# B&R Automation Studio project lab3
Automation Studio 

## Configuration Real

CPU 4PP065.0571-P74, AutomationRuntime D4.52, Build 4.1.2, Vc V4.52.0, Safety 1.6

### Task classes (Cpu.sw)
```
Cyclic#1 (cycle 2000 us, tolerance 0 us):
  ncsdcctrl <- ncsdcctrl.prg
  SDCAxisCtr <- SDCAxisCtrl_X.prg
  SDCAxisCt2 <- SDCAxisCtrl_Z.prg
  SDCAxisCt1 <- SDCAxisCtrl_Y.prg
Cyclic#2:
  User_Inter <- User_Interface.prg
DataObjects: Arnc0sys, Acp10sys
NcDataObjects: AxisInit <- AxisInit.dob, gAxis03a <- gAxis03obj.gAxis03a.dob, gAxis03i <- gAxis03obj.gAxis03i.dob, AxisApt <- AxisApt.dob, gmcipsys <- GmcIpConfig.gmcipsys.dob, gmcipusm <- GmcIpUserConfig.gmcipusm.dob, gmciplbr <- GmcIpConfig.gmciplbr.dob, gmcipvar <- GmcIpUserConfig.gmcipvar.dob, gmcipcbr <- GmcIpConfig.gmcipcbr.dob, gmcipubr <- GmcIpUserConfig.gmcipubr.dob, gmciplsm <- GmcIpConfig.gmciplsm.dob, gmcipui <- GmcIpUserConfig.gmcipui.dob, gmcipcsm <- GmcIpConfig.gmcipcsm.dob, gmcipuc <- GmcIpUserConfig.gmcipuc.dob, gmcipcfg <- GmcIpConfig.gmcipcfg.dob, gmcipfub <- GmcIpUserConfig.gmcipfub.dob, gmcipiec <- GmcIpConfig.gmcipiec.dob, gmcipus <- GmcIpUserConfig.gmcipus.dob, gmciplog <- GmcIpConfig.gmciplog.dob, gmcipfun <- GmcIpUserConfig.gmcipfun.dob, gmcipesm <- GmcIpConfig.gmcipesm.dob, gmcipmxd <- GmcIpConfig.gmcipmxd.dob, gmcipmx <- GmcIpConfig.gmcipmx.dob, CncInit <- CncInit.dob, CncProg1 <- CncProg1.dob, CncProg <- CncProg.dob
VcDataObjects: Visu <- Visu.dob
Binaries: TCData, vccbtn, arialbd, vcmgr, vcfile, vccnum, vcpfpp30, vcfntttf, vctcal, vcdsloc, vcgclass, vcpfmtcx, vcbclass, udbdef, arial, Visu03, vcalarm, Visu01, vcptelo, vcpdpp30, vcrt, vcshared, Visu02, vcctext, vcdsint, vcpdsw, vccovl, arconfig, User, Role, sysconf, iomap, asfw, ashwd, ashwac, Acp10map1, acp10cfg, Acp10map, arnc0cfg, Arnc0map
Libraries: Acp10sdc, Library, Acp10man, Acp10_MC, sys_lib, brsystem, asstring, AsMath, Arnc0man, DataObj, AsArLog, FileIO, AsArProf, AsMem, Runtime, astime, Acp10par, NcGlobal, Acp10sim, powerlnk, asieccon, asiotime, vcresman, operator
```

### Hardware
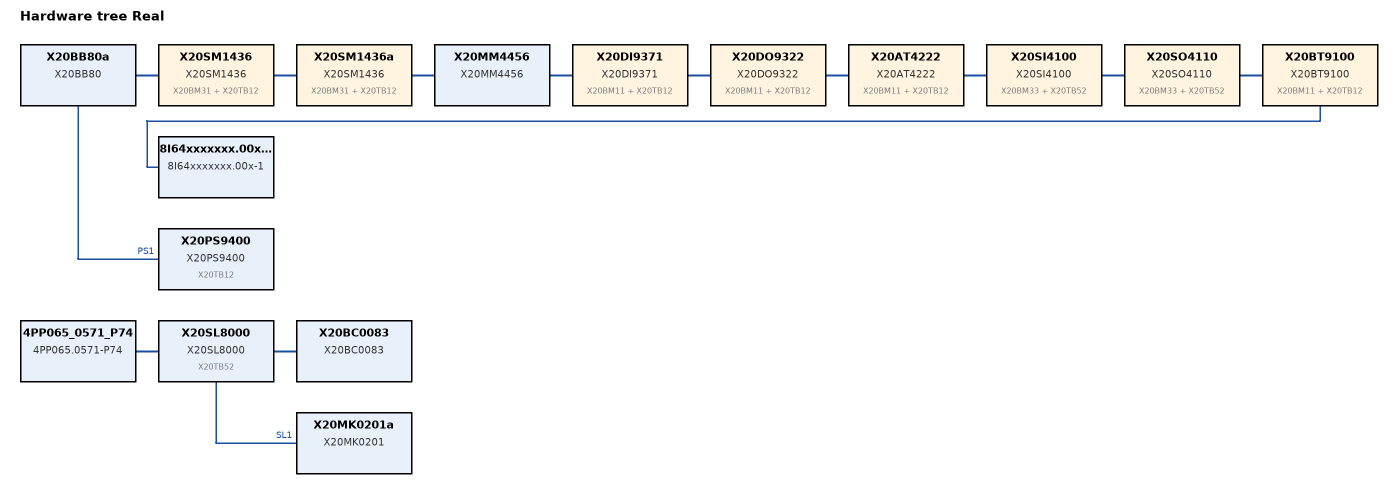
```
4PP065_0571_P74 : 4PP065.0571-P74 v1.1.2.0
  Connector IF4:
    Channel1
    ChannelID1 = McAcpBroadcast
    ChannelType1 = OCTET[96]
  Connector IF5:
    ActivateDevice = 1
    Mode = Manual
    InternetAddress = 10.0.1.14
    SubnetMask = 255.255.255.0
  ConfigurationID = labBR
  TimerDeviceType = EPLX2X
  TimerDevice = 4PP065_0571_P74.IF4
  TaskClassIdleTime = 2000
  Cyclic1Duration = 2000
  Cyclic1Tolerance = 0
  Cyclic1Output = 1
  Cyclic3Tolerance = 0
  VcObjectName = Visu
8I64xxxxxxx.00x-1 : 8I64xxxxxxx.00x-1 v1.3.9.1  [X2X1 -> X20BT9100.X2X1 [Cable Type=X2XCable, Length=10, Version=1.0.0.2]]
  BothEndSwitchesAreNormallyOpen_r1 = on
  QuickStopIsNormallyOpen_r1 = on
X20AT4222 : X20AT4222 v1.2.3.0  [SS1 -> X20TB12f.SS; SL -> X20BM11c.SL1]
X20BB80a : X20BB80 v1.0.2.0
X20BC0083 : X20BC0083 v2.7.0.0  [PLK1 -> X20SL8000.PLK2 (NodeNumber=2) [Cable Type=PowerlinkCable, Length=10, Version=1.0.0.2]; SL -> X20BB80a.SL1]
X20BM11a : X20BM11 v1.0.0.1  [X2X1 -> X20MM4456.X2X2]
X20BM11b : X20BM11 v1.0.0.1  [X2X1 -> X20BM11a.X2X2]
X20BM11c : X20BM11 v1.0.0.1  [X2X1 -> X20BM11b.X2X2]
X20BM11d : X20BM11 v1.0.0.1  [X2X1 -> X20BM33b.X2X2]
X20BM31a : X20BM31 v1.0.0.1  [X2X1 -> X20BB80a.IF1]
X20BM31b : X20BM31 v1.0.0.1  [X2X1 -> X20BM31a.X2X2]
X20BM33a : X20BM33 v1.0.0.4  [X2X1 -> X20BM11c.X2X2]
X20BM33b : X20BM33 v1.0.0.4  [X2X1 -> X20BM33a.X2X2]
X20BT9100 : X20BT9100 v1.0.3.0  [SS1 -> X20TB12g.SS; SL -> X20BM11d.SL1]
X20DI9371 : X20DI9371 v1.0.2.0  [SS1 -> X20TB12d.SS; SL -> X20BM11a.SL1]
X20DO9322 : X20DO9322 v1.0.3.0  [SS1 -> X20TB12e.SS; SL -> X20BM11b.SL1]
X20MK0201a : X20MK0201 v1.0.0.0 (Disabled=true)  [SL -> X20SL8000.SL1]
X20MM4456 : X20MM4456 v1.1.5.0  [X2X1 -> X20BM31b.X2X2]
X20PS9400 : X20PS9400 v1.0.2.4  [SS1 -> X20TB12b.SS; PS -> X20BB80a.PS1]
X20SI4100 : X20SI4100 v1.10.1.1  [SS1 -> X20TB52b.SS; SL -> X20BM33a.SL1]
X20SL8000 : X20SL8000 v1.6.5.1 (Disabled=true)  [PLK1 -> 4PP065_0571_P74.IF4 (NodeNumber=1) [Cable Type=PowerlinkCable, Length=10, Version=1.0.0.2]; PLK2 -> X20BC0083.PLK1 (NodeNumber=1) [Cable Type=PowerlinkCable, Length=10, Version=1.0.0.2]; SS1 -> X20TB52a.SS]
  SafeProject = SafeLOGIC-1
X20SM1436 : X20SM1436 v1.4.2.1  [SS1 -> X20TB12a.SS; SL -> X20BM31a.SL1]
X20SM1436a : X20SM1436 v1.4.2.1  [SS1 -> X20TB12c.SS; SL -> X20BM31b.SL1]
X20SO4110 : X20SO4110 v1.10.1.1  [SS1 -> X20TB52c.SS; SL -> X20BM33b.SL1]
  SafeLogicID = 2
  SafeModuleID = 3
X20TB12a : X20TB12 v1.0.0.0
X20TB12b : X20TB12 v1.0.0.0
X20TB12c : X20TB12 v1.0.0.0
X20TB12d : X20TB12 v1.0.0.0
X20TB12e : X20TB12 v1.0.0.0
X20TB12f : X20TB12 v1.0.0.0
X20TB12g : X20TB12 v1.0.0.0
X20TB52a : X20TB52 v1.0.0.1 (Disabled=true)
X20TB52b : X20TB52 v1.0.0.1
X20TB52c : X20TB52 v1.0.0.1
```

## Configuration Simulation

### Task classes (Cpu.sw)
```
Cyclic#1:
  SDCAxisCtr <- SDCAxisCtrl_X.prg
DataObjects: Acp10sys
NcDataObjects: AxisApt <- AxisApt.dob, AxisInit <- AxisInit.dob, acp10etxen <- acp10etxen.dob
Binaries: TCData, ashwd, sysconf, asfw, arconfig, iomap, Acp10map, Acp10map1, arnc0cfg, acp10cfg
Libraries: AsIecCon, astime, Acp10sdc, Acp10man, Acp10par, NcGlobal, asstring, AsIOTime, Acp10_MC, brsystem, sys_lib, Runtime, Acp10sim, fileio, powerlnk, Library
```

## Logical view

Binary libraries used (declarations not repeated): Runtime, Operator, AsIecCon, astime, asstring, AsIOTime, brsystem, sys_lib, AsMath, DataObj, AsArLog, FileIO, AsArProf, AsMem, Acp10man, Acp10par, NcGlobal, Acp10sim, Acp10_MC, Acp10sdc, Arnc0man 5.02.1

### Global.var
```iecst
VAR
	Trajectory : FB_Trajectory := (0); (*Переменная типа Функциональный блок управления УРТК*)
	Move_axis : FB_move := (0); (*Переменная типа Функциональный блок движения оси*)
	Power_home : FB_power := (0); (*Переменная типа Функциональный блок запуска и референсирование осей*)
	AxisX : ACP10AXIS_typ := (0); (*Ось X*)
	AxisX_EncIf : SdcEncIf16_typ := (0);
	AxisX_DrvIf : SdcDrvIf16_typ := (0);
	AxisX_DiDoIf : SdcDiDoIf_typ := (0);
	AxisX_HW : SdcHwCfg_typ := (0);
	AxisY : ACP10AXIS_typ := (0); (*Ось Y*)
	AxisY_EncIf : SdcEncIf16_typ := (0);
	AxisY_DrvIf : SdcDrvIf16_typ := (0);
	AxisY_DiDoIf : SdcDiDoIf_typ := (0);
	AxisY_HW : SdcHwCfg_typ := (0);
	AxisZ : ACP10AXIS_typ := (0); (*Ось Z*)
	AxisZ_EncIf : SdcEncIf16_typ := (0);
	AxisZ_DrvIf : SdcDrvIf16_typ := (0);
	AxisZ_DiDoIf : SdcDiDoIf_typ := (0);
	AxisZ_HW : SdcHwCfg_typ := (0);
	gAxis01 : ACP10AXIS_typ := (0);
	gAxis02 : ACP10AXIS_typ := (0);
	gAxisTest : ACP10AXIS_typ := (0);
	gAxisTest_HW : SdcHwCfg_typ := (0);
	gAxisTest_DrvIf : SdcDrvIf16_typ := (0);
	gAxisTest_DiDoIf : SdcDiDoIf_typ := (0);
	gAxisTest_ModuleOk : BOOL := 0;
	gAxis03 : ACP10AXIS_typ := (0);
	gAxis03_HW : SdcHwCfg_typ := (0);
	gAxis03_DrvIf : SdcDrvIf16_typ := (0);
	gAxis03_DiDoIf : SdcDiDoIf_typ := (0);
	gAxis03_ModuleOk : BOOL := 0;
	CNCsys : ARNC0CNC_typ;
END_VAR
```

### AxInitAcp10.ax
```
InitParameter (Version=5.2.1, NcSwId=ACP10)
  ACP10AXIS_typ:
    dig_in:
      level:
        reference = ncACTIV_HI
        pos_hw_end = ncACTIV_HI
        neg_hw_end = ncACTIV_HI
        trigger1 = ncACTIV_HI
        trigger2 = ncACTIV_HI
    encoder_if:
      parameter:
        count_dir = ncSTANDARD
        scaling:
          load:
            units = 3000
            rev_motor = 1
    limit:
      parameter:
        v_pos = 7500.0
        v_neg = 7500.0
        a1_pos = 10000.0
        a2_pos = 10000.0
        a1_neg = 10000.0
        a2_neg = 10000.0
        t_jolt = 0.0
        t_in_pos = 0.0
        pos_sw_end = 8388607
        neg_sw_end = -8388608
        ds_warning = 500.0
        ds_stop = 1000.0
        a_stop = 1.0E+30
        dv_stop = 0.0
        dv_stop_mode = ncOFF
    controller:
      mode = ncPOSITION
      position:
        kv = 10.0
        tn = 0.0
        t_predict = 0.04
        t_total = 0.04
        p_max = 10000.0
        i_max = 0.0
      speed:
        kv = 100.0
        tn = 0.04
        t_filter = 0.0
        isq_filter1:
          type = ncOFF
          a0 = 0.0
          a1 = 0.0
          b0 = 0.0
          b1 = 0.0
          b2 = 0.0
          c0_par_id = 0
          c1_par_id = 0
        isq_filter2:
          type = ncOFF
          a0 = 0.0
          a1 = 0.0
          b0 = 0.0
          b1 = 0.0
          b2 = 0.0
          c0_par_id = 0
          c1_par_id = 0
        isq_filter3:
          type = ncOFF
          a0 = 0.0
          a1 = 0.0
          b0 = 0.0
          b1 = 0.0
          b2 = 0.0
          c0_par_id = 0
          c1_par_id = 0
      uf:
        type = ncLINEAR
        auto_config = ncMOTOR_PAR
        u0 = 0.0
        un = 0.0
        fn = 50.0
        k_f_slip = 0.0
      ff:
        torque_load = 0.0
        torque_pos = 0.0
        torque_neg = 0.0
        kv_torque = 0.0
        inertia = 0.0
        t_filter_a = 0.0
    move:
      stop:
        parameter[0]:
          decel_ramp = ncA_LIMIT
          controller = ncON
        parameter[1]:
          decel_ramp = ncA_LIMIT
          controller = ncON
        parameter[2]:
          decel_ramp = ncA_LIMIT
          controller = ncON
        parameter[3]:
          decel_ramp = ncA_LIMIT
          controller = ncON
        quickstop:
          decel_ramp = ncA_LIMIT
          t_jolt = 0.0
        drive_error:
          decel_ramp = ncA_LIMIT
      homing:
        parameter:
          s = 0
          v_switch = 2000.0
          v_trigger = 1000.0
          a = 5000.0
          mode = ncDIRECT
          edge_sw = ncNEGATIVE
          start_dir = ncPOSITIVE
          trigg_dir = ncNEGATIVE
          ref_pulse = ncOFF
          fix_dir = ncOFF
          tr_s_block = 0.0
          torque_lim = 0.0
          ds_block = 0.0
          ds_stop = 0.0
      basis:
        parameter:
          v_pos = 6000.0
          v_neg = 6000.0
          a1_pos = 12000.0
          a2_pos = 12000.0
          a1_neg = 12000.0
          a2_neg = 12000.0
    message:
      text:
        parameter:
          format = ncBREAK
          columns = 80
          data_modul
```

- Data object Logical/CncInit (Cns) (no source held here)

- Data object Logical/CncProg (Cnc) (no source held here)

- Data object Logical/GmcIpConfig/gmcipsys (Cnc, version 5.02.1) (no source held here)

- Data object Logical/GmcIpConfig/gmciplbr (Cnc, version 5.02.1) (no source held here)

- Data object Logical/GmcIpConfig/gmcipcbr (Cnc, version 5.02.1) (no source held here)

- Data object Logical/GmcIpConfig/gmciplsm (Cnc, version 5.02.1) (no source held here)

- Data object Logical/GmcIpConfig/gmcipcsm (Cnc, version 5.02.1) (no source held here)

- Data object Logical/GmcIpConfig/gmcipcfg (Cnc, version 5.02.1) (no source held here)

- Data object Logical/GmcIpConfig/gmcipiec (Cnc, version 5.02.1) (no source held here)

- Data object Logical/GmcIpConfig/gmciplog (Cnc, version 5.02.1) (no source held here)

- Data object Logical/GmcIpConfig/gmcipesm (Cnc, version 5.02.1) (no source held here)

- Data object Logical/GmcIpConfig/gmcipmxd (Cnc, version 5.02.1) (no source held here)

- Data object Logical/GmcIpConfig/gmcipmx (Cnc, version 5.02.1) (no source held here)

- Data object Logical/GmcIpUserConfig/gmcipfub (Cnc, version 5.02.1) (no source held here)

- Data object Logical/GmcIpUserConfig/gmcipfun (Cnc, version 5.02.1) (no source held here)

- Data object Logical/GmcIpUserConfig/gmcipubr (Cnc, version 5.02.1) (no source held here)

- Data object Logical/GmcIpUserConfig/gmcipuc (Cnc, version 5.02.1) (no source held here)

### Library Logical/Libraries/Library (ANSIC)
Depends on: Runtime, Operator, AsIecCon, astime, asstring, AsIOTime, brsystem, sys_lib, AsMath, DataObj, AsArLog, FileIO, AsArProf, AsMem, Acp10man, Acp10par, NcGlobal, Acp10sim, Acp10_MC, Acp10sdc, Arnc0man

#### Types.typ
```iecst
TYPE
	T_State_Trajectory :
		(
		Idle_Trajectory,
		Done_Trajectory,
		side1,
		side2,
		side3,
		side4,
		PowerY,
		PowerZ,
		Stop_Trajectory
		);
	T_State_move :
		(
		Idle_move,
		Move,
		Done_move
		);
	T_State_power :
		(
		Idle,
		Power,
		Home,
		Done
		);
END_TYPE
```

#### Library.fun
```iecst
FUNCTION_BLOCK FB_Motor (*TODO: Add your comment here*) (*$GROUP=User,$CAT=User,$GROUPICON=User.png,$CATICON=User.png*)
	VAR_INPUT
		in : REAL;
	END_VAR
	VAR_OUTPUT
		out_w : REAL;
		out_phi : REAL;
	END_VAR
	VAR
		k_e : REAL;
		T_m : REAL;
		dt : REAL;
		integrator : FB_Integrator;
		integrator_phi : FB_Integrator;
	END_VAR
END_FUNCTION_BLOCK

FUNCTION_BLOCK FB_Integrator (*TODO: Add your comment here*) (*$GROUP=User,$CAT=User,$GROUPICON=User.png,$CATICON=User.png*)
	VAR_INPUT
		in : REAL;
		dt : REAL;
	END_VAR
	VAR_OUTPUT
		out : REAL;
	END_VAR
	VAR
		state : REAL := 0.0;
	END_VAR
END_FUNCTION_BLOCK

FUNCTION_BLOCK FB_Controller (* *) (*$GROUP=User,$CAT=User,$GROUPICON=User.png,$CATICON=User.png*)
	VAR_INPUT
		in : REAL;
	END_VAR
	VAR_OUTPUT
		out : REAL;
	END_VAR
	VAR
		k_i : REAL;
		sum : REAL;
		k_p : REAL;
		dt : REAL;
		max_abs_value : REAL;
		integrator : FB_Integrator;
		last_sum : REAL;
	END_VAR
END_FUNCTION_BLOCK

FUNCTION_BLOCK FB_Endswitch (*TODO: Add your comment here*) (*$GROUP=User,$CAT=User,$GROUPICON=User.png,$CATICON=User.png*)
	VAR_INPUT
		in : REAL;
		neg_value : REAL;
		pos_value : REAL;
	END_VAR
	VAR_OUTPUT
		neg_reached : BOOL;
		pos_reached : BOOL;
	END_VAR
END_FUNCTION_BLOCK

FUNCTION_BLOCK FB_Axis (*TODO: Add your comment here*) (*$GROUP=User,$CAT=User,$GROUPICON=User.png,$CATICON=User.png*)
	VAR_INPUT
		reset_error : BOOL;
		endswitch_a_reached : BOOL;
		endswitch_b_reached : BOOL;
		pwm_percentage : SINT;
	END_VAR
	VAR_OUTPUT
		reset_counter : BOOL;
		pwm_value : INT;
	END_VAR
	VAR_OUTPUT RETAIN
		counter : INT;
	END_VAR
	VAR_OUTPUT
		speed : REAL;
	END_VAR
	VAR
		last_counter : INT;
	END_VAR
END_FUNCTION_BLOCK

{REDUND_ERROR} FUNCTION_BLOCK FB_power (*Функциональный блок запуска и референсирование осей*) (*$GROUP=User,$CAT=User,$GROUPICON=User.png,$CATICON=User.png*)
	VAR_INPUT
		State : T_State_power;
		Power : MC_Power;
		Home : MC_Home;
		Axis : UDINT;
		enable : BOOL;
	END_VAR
	VAR_OUTPUT
		done : BOOL;
	END_VAR
END_FUNCTION_BLOCK

{REDUND_ERROR} FUNCTION_BLOCK FB_move (*Функциональный блок движения оси*) (*$GROUP=User,$CAT=User,$GROUPICON=User.png,$CATICON=User.png*)
	VAR_INPUT
		Axis : UDINT;
		enable : BOOL;
		Move : MC_MoveAdditive;
		length : REAL;
	END_VAR
	VAR_OUTPUT
		done : BOOL;
	END_VAR
	VAR
		State : T_State_move;
	END_VAR
END_FUNCTION_BLOCK

{REDUND_ERROR} FUNCTION_BLOCK FB_Trajectory (*Функциональный блок управления УРТК*) (*$GROUP=User,$CAT=User,$GROUPICON=User.png,$CATICON=User.png*)
	VAR_INPUT
		enable : BOOL;
		AxisY : UDINT;
		AxisZ : UDINT;
		length : REAL;
	END_VAR
	VAR_OUTPUT
		done : BOOL;
	END_VAR
	VAR
		State : T_State_Trajectory;
		Power_AxisY : FB_power;
		Power_AxisZ : FB_power;
		Move_Axis : FB_move;
	END_VAR
END_FUNCTION_BLOCK
```

#### FB_Motor.c
```c
#include <bur/plctypes.h>
#ifdef __cplusplus
	extern "C"
	{
#endif
	#include "Library.h"
#ifdef __cplusplus
	};
#endif
/* TODO: Add your comment here */
void FB_Motor(struct FB_Motor* inst)
{
	REAL a = inst->in / inst->k_e - inst->out_w;
	REAL b = a / inst->T_m;
	inst->integrator.dt = inst->dt;
	inst->integrator_phi.dt = inst->dt;
	inst->integrator.in = b;
	FB_Integrator(&inst->integrator);
	inst->out_w = inst->integrator.out;
	inst->integrator_phi.in = inst->out_w;
	FB_Integrator(&inst->integrator_phi);
	inst->out_phi = inst->integrator_phi.out;
}
```

#### FB_Controller.c
```c
#include <bur/plctypes.h>
#ifdef __cplusplus
	extern "C"
	{
#endif
	#include "Library.h"
#ifdef __cplusplus
	};
#endif

void FB_Controller(struct FB_Controller* inst)
{
	REAL a = inst->in * inst->k_p;
	REAL b = inst->in * inst->k_i;
	inst->integrator.dt = inst->dt;
	inst->integrator.in = b;
	FB_Integrator(&inst->integrator);
	a = a > inst->max_abs_value ? inst->max_abs_value : a;
	a = a < -inst->max_abs_value ? -inst->max_abs_value : a;
	inst->sum = a + inst->integrator.out;
	inst->out = inst->sum;
	inst->out = inst->out > inst->max_abs_value ? inst->max_abs_value : inst->out;
	inst->out = inst->out < -inst->max_abs_value ? -inst->max_abs_value : inst->out;
	inst->last_sum = (inst->out - inst->sum);
	inst->integrator.state = inst->integrator.state + inst->last_sum;
}
```

#### FB_Endswitch.c
```c
#include <bur/plctypes.h>
#ifdef __cplusplus
	extern "C"
	{
#endif
	#include "Library.h"
#ifdef __cplusplus
	};
#endif
/* TODO: Add your comment here */
void FB_Endswitch(struct FB_Endswitch* inst)
{
	inst->pos_reached = inst->in >= inst->pos_value ? 1 : 0;
	inst->neg_reached = inst->in <= inst->neg_value ? 1 : 0;
}
```

#### FB_Axis.c
```c
#include <bur/plctypes.h>
#ifdef __cplusplus
	extern "C"
	{
#endif
	#include "Library.h"
#ifdef __cplusplus
	};
#endif
/* TODO: Add your comment here */
void FB_Axis(struct FB_Axis* inst)
{
	/*
	if (inst->pwm_percentage > 100)
	{
		inst->pwm_percentage = 100;
	}
	if (inst->pwm_percentage < -100)
	{
		inst->pwm_percentage = -100;
	}
	REAL raw_percentage = (REAL) inst->pwm_percentage / 100.0 * 32767.0;
	inst->pwm_value = (INT) raw_percentage;
	*/
	inst->speed = inst->counter - inst->last_counter;
	inst->speed = (inst->speed * 3000 / 24.0) / 0.002;
	inst->last_counter = inst->counter;
}
```

#### FB_power.c
```c
#include <bur/plctypes.h>
#ifdef __cplusplus
	extern "C"
	{
#endif
	#include "Library.h"
#ifdef __cplusplus
	};
#endif
/* TODO: Add your comment here */
void FB_power(struct FB_power* inst) // Функциональный блок запуска и референсирования осей
{
	switch (inst->State) // Машина состояний для ФБ
	{
		case Idle: // Состояние покоя
			{
				if(inst->enable)
				{
					inst->done = 0;
					inst->State = Power; // Переход к состоянию запуска
				}

				break;
			}
		case Power: // Состояние запуска
			{
				inst->Power.Axis = inst->Axis;
				inst->Power.Enable = 1;

				inst->State = Home; // Переход к состоянию референсирования

				break;
			}
		case Home: // Состояние референсирования осей
			{
				inst->Home.Axis = inst->Axis;
				inst->Home.Execute = 1;
				inst->Home.HomingMode = 1;
				inst->Home.Position = 0;
				if (inst->Home.Done)
				{
					inst->State = Done; // Переход к состоянию завершения
				}

				break;
			}
		case Done: // Состояние завершения работы
			{
				inst->done = 1;
				if(inst->done)
				{
					inst->Home.Done = 0;
					inst->enable = 0;
					inst->State = Idle; // Переход в состояние покоя после завершения
				}

				break;
			}
	}

	//Инициализация использованных функциональных блоков
	MC_Power(&inst->Power);
	MC_Home(&inst->Home);

}
```

#### FB_move.c
```c
#include <bur/plctypes.h>
#ifdef __cplusplus
	extern "C"
	{
#endif
	#include "Library.h"
#ifdef __cplusplus
	};
#endif
/* TODO: Add your comment here */
void FB_move(struct FB_move* inst) // Функциональный блок движения оси
{
	switch (inst->State) // Машина состояний
	{
		case Idle_move: // Состояние покоя
			{
				if(inst->enable)
				{
					inst->Move.Done = 0;
					inst->done = 0;
					inst->State = Move; // Переход к состоянию движения
				}

				break;
			}
		case Move: // Состояние движение
			{
				// Передача необходимых параметров в функциональный блок
				inst->Move.Axis = inst->Axis;
				inst->Move.Execute = 1;
				inst->Move.Distance = inst->length;
				inst->Move.Velocity = 3000;
				inst->Move.Acceleration = 6000;
				inst->Move.Deceleration = 6000;

				if(inst->Move.Done)
				{
					inst->State = Done_move; // Переход к состоянию завершения
				}

				break;
			}
		case Done_move: // Состояние завершения
			{
				inst->done = 1;
				if(inst->done)
				{
					inst->Move.Execute = 0;
					inst->length = 0;
					inst->enable = 0;
					inst->State = Idle_move;
				}

				break;
			}
	}
	MC_MoveAdditive(&inst->Move); // Инициализация Функционального блока движения
}
//ВсеГО хорошеГО
```

#### FB_Trajectory.c
```c
#include <bur/plctypes.h>
#ifdef __cplusplus
	extern "C"
	{
#endif
	#include "Library.h"
#ifdef __cplusplus
	};
#endif
/* TODO: Add your comment here */
void FB_Trajectory(struct FB_Trajectory* inst) // Функциональный блок управления УРТК
{
	switch (inst->State) // Машина состояний
	{
		case Idle_Trajectory: // Состояние покоя
			{
				if (inst->enable)
				{
					inst->done = 0;
					inst->State = PowerY; // Переход к запуску оси Y
				}
				break;
			}
		case PowerY : // Запуск оси Y
			{
				inst->Power_AxisY.Axis = inst->AxisY; // Объявление оси Y
				inst->Power_AxisY.enable = 1;
				if(inst->Power_AxisY.done)
				{
					inst->State = PowerZ; // Переход к запуску оси Z
				}
				break;
			}
		case PowerZ :  // Запуск оси Z
			{
				inst->Power_AxisZ.Axis = inst->AxisZ; // Объявление оси Z
				inst->Power_AxisZ.enable = 1;
				if(inst->Power_AxisZ.done)
				{
					inst->State = side1; // Переход к состоянию движения по траектории 1-й стороны
				}
				break;
			}
		case side1 : // Состояние движения по траектории 1-й стороны
			{
				inst->Move_Axis.Axis = inst->AxisY;
				inst->Move_Axis.length = inst->length*100;
				inst->Move_Axis.enable = 1;
				if(inst->Move_Axis.done)
				{
					inst->State = side2; // Переход к состоянию движения по траектории 2-й стороны
				}
				break;
			}
		case side2 : // Состояние движения по траектории 2-й стороны
			{
				inst->Move_Axis.Axis = inst->AxisZ;
				inst->Move_Axis.length = inst->length*100;
				inst->Move_Axis.enable = 1;
				if(inst->Move_Axis.done)
				{
					inst->State = side3; // Переход к состоянию движения по траектории 3-й стороны
				}
				break;
			}
		case side3 : // Состояние движения по траектории 3-й стороны
			{
				inst->Move_Axis.Axis = inst->AxisY;
				inst->Move_Axis.length = -inst->length*100;
				inst->Move_Axis.enable = 1;
				if(inst->Move_Axis.done)
				{
					inst->State = side4; // Переход к состоянию движения по траектории 4-й стороны
				}
				break;
			}
		case side4 : // Состояние движения по траектории 4-й стороны
			{
				inst->Move_Axis.Axis = inst->AxisZ;
				inst->Move_Axis.length = -inst->length*100;
				inst->Move_Axis.enable = 1;
				if(inst->Move_Axis.done)
				{
					inst->State = Stop_Trajectory; // Переход к состоянию остановки и выключения УРТК
				}
				break;
			}
		case Stop_Trajectory : // Состояние остановке и выключения УРТК
			{
				inst->Power_AxisY.Power.Enable = 0;
				inst->Power_AxisZ.Power.Enable = 0;
				if (!inst->Power_AxisY.Power.Status && !inst->Power_AxisZ.Power.Status)
				{
					inst->State = Done_Trajectory; // Переход к состоянию завершения работы ФБ
				}
			}
		case Done_Trajectory : // Состояние завершения работы ФБ
			{
				inst->done = 1;
				if(inst->done)
				{
					inst->Move_Axis.done = 0;
					inst->Move_Axis.done = 0;
					inst->enable = 0;
					inst->State = Idle_Trajectory;
				}
				break;
			}
	}

	// Инициализация использованных функциональных блоков
	FB_move(&inst->Move_Axis);
	FB_power(&inst->Power_AxisY);
	FB_power(&inst->Power_AxisZ);
}
```

Listed in the project but not available here: Logical/Libraries/Library/FB_Integrator.c
